(* IEC 61131-3 sources: CodesysTest/alpha/export/FBs/Motors/Festo/FB_FestoMotor.pou/Homing.prop, 1 file *)

(* ---- Get.pm.st ---- *)
(*#-#-#-#-#-#-#-#-#-#---Declaration---#-#-#-#-#-#-#-#-#-#-#-#-#*)

VAR
END_VAR
(*#-#-#-#-#-#-#-#-#-#---Implementation---#-#-#-#-#-#-#-#-#-#-#-#-#*)

Homing := homingActive;
